{attribute 'GeneratedUsingTerminal: EK1122-0000-0018'}
{attribute addProperty BoxType "EK1122-0000-0018"}
{attribute addProperty Id "Beckhoff_EKM1xxxsub_EK1100EK1100_AB5A94672A_0001_EKM1101_0000_0016EKM1101_B1409E5482A_0002_EKM1101_0000_0017EKM1101_B1409E5482A_0003_EKM1101_0000_0018EKM1101_B1409E5482A_0004_EKM1101_0000_0019EKM1101_B1409E5482A_0005_EKM1101_0000_0020EKM1101_B1409E5482"}
{attribute addProperty CRC "1764167585"}
{attribute addProperty Size "412"}
TYPE Beckhoff_EKM1xxxEK1122_69270FA1 EXTENDS EK1122_AB5A9467 :
STRUCT
	{attribute addProperty Name "Beckhoff_EKM1xxxsub_EK1100"}
	Beckhoff_EKM1xxxsub_EK1100 : EK1100_AB5A9467;
	{attribute addProperty Name "A_0001_EKM1101_0000_0016"}
	A_0001_EKM1101_0000_0016 : EKM1101_B1409E54;
	{attribute addProperty Name "A_0002_EKM1101_0000_0017"}
	A_0002_EKM1101_0000_0017 : EKM1101_B1409E54;
	{attribute addProperty Name "A_0003_EKM1101_0000_0018"}
	A_0003_EKM1101_0000_0018 : EKM1101_B1409E54;
	{attribute addProperty Name "A_0004_EKM1101_0000_0019"}
	A_0004_EKM1101_0000_0019 : EKM1101_B1409E54;
	{attribute addProperty Name "A_0005_EKM1101_0000_0020"}
	A_0005_EKM1101_0000_0020 : EKM1101_B1409E54;
END_STRUCT
END_TYPE

(* stored: Version 1.2.0.0, ProductVersion 3.1.4024.9
   DUT Beckhoff_EKM1xxxEK1122_69270FA1: Id {dfe41db2-34e0-460a-b68c-bc4e18458b62} *)
